INTERFACE I_Subject

METHOD Attach : BOOL
VAR_INPUT
	ipObserver		: I_Observer;
END_VAR
END_METHOD

METHOD Detach : BOOL
VAR_INPUT	
	ipObserver		: I_Observer;
END_VAR
END_METHOD

END_INTERFACE

(* stored: Version 1.1.0.1, ProductVersion 3.1.4022.7
   Itf I_Subject: Id {6890b304-c5dc-46c3-9482-198f619d2f56}
   Method Attach: Id {62711a66-5623-4145-ad91-ad84aea7c33f}
   Method Detach: Id {4393bf18-6fd0-421d-a34a-3458d26e55fe} *)
